TYPE Kickout_Inputs_typ:
STRUCT
	BallClampOpened AT %I*: BOOL;
	BallClampClosed AT %I*: BOOL;
	BallRemoved AT %I*: BOOL;
END_STRUCT
END_TYPE

(* stored: Version 1.1.0.1, ProductVersion 3.1.4024.12
   DUT Kickout_Inputs_typ: Id {56fda4c3-4363-0dc1-106c-9ddc2e44e1c7} *)
